{attribute 'GeneratedUsingTerminal: EK1100-0000-0018'}
{attribute addProperty BoxType "EK1100-0000-0018"}
{attribute addProperty Id "RP20_A2_EK1122RP20_A2_EK1122_68D808EA135RP20_A4_EL7041_1000EL7041_86DE63E743RP20_A5_EL7041_1000EL7041_86DE63E743RP20_A6_EL1809EL1809_32157CFD20RP20_A7_EL2809EL2809_2B6483BD19RP20_EndTerminal_EL9011EL9011_D65D3D320"}
{attribute addProperty CRC "2049168895"}
{attribute addProperty Size "260"}
{attribute addProperty Name "RP20 (EK1100)"}
TYPE RP20_EK1100_7A23D5FF EXTENDS EK1100_1FC0878B :
STRUCT
	{attribute addProperty Name "RP20_A2 (EK1122)"}
	{attribute addProperty PreviousPort "RP20 (EK1100) : B"}
	{attribute addProperty SyncUnit "default"}
	RP20_A2_EK1122 : RP20_A2_EK1122_68D808EA;
	{attribute addProperty Name "RP20_A4 (EL7041-1000)"}
	{attribute addProperty PreviousPort "RP20_A2 (EK1122) : C"}
	{attribute addProperty SyncUnit "P20"}
	RP20_A4_EL7041_1000 : EL7041_86DE63E7;
	{attribute addProperty Name "RP20_A5 (EL7041-1000)"}
	{attribute addProperty PreviousPort "RP20_A4 (EL7041-1000) : B"}
	{attribute addProperty SyncUnit "P20"}
	RP20_A5_EL7041_1000 : EL7041_86DE63E7;
	{attribute addProperty Name "RP20_A6 (EL1809)"}
	{attribute addProperty PreviousPort "RP20_A5 (EL7041-1000) : B"}
	{attribute addProperty SyncUnit "P20"}
	RP20_A6_EL1809 : EL1809_32157CFD;
	{attribute addProperty Name "RP20_A7 (EL2809)"}
	{attribute addProperty PreviousPort "RP20_A6 (EL1809) : B"}
	{attribute addProperty SyncUnit "P20"}
	RP20_A7_EL2809 : EL2809_2B6483BD;
	{attribute addProperty Name "RP20_EndTerminal (EL9011)"}
	{attribute addProperty PreviousPort "RP20_A7 (EL2809) : B"}
	{attribute addProperty SyncUnit "default"}
	RP20_EndTerminal_EL9011 : EL9011_D65D3D32;
END_STRUCT
END_TYPE

(* stored: Version 1.2.0.0, ProductVersion 3.1.4024.11
   DUT RP20_EK1100_7A23D5FF: Id {5bd3e28d-7b31-0552-3ee5-9538c6400c14} *)
